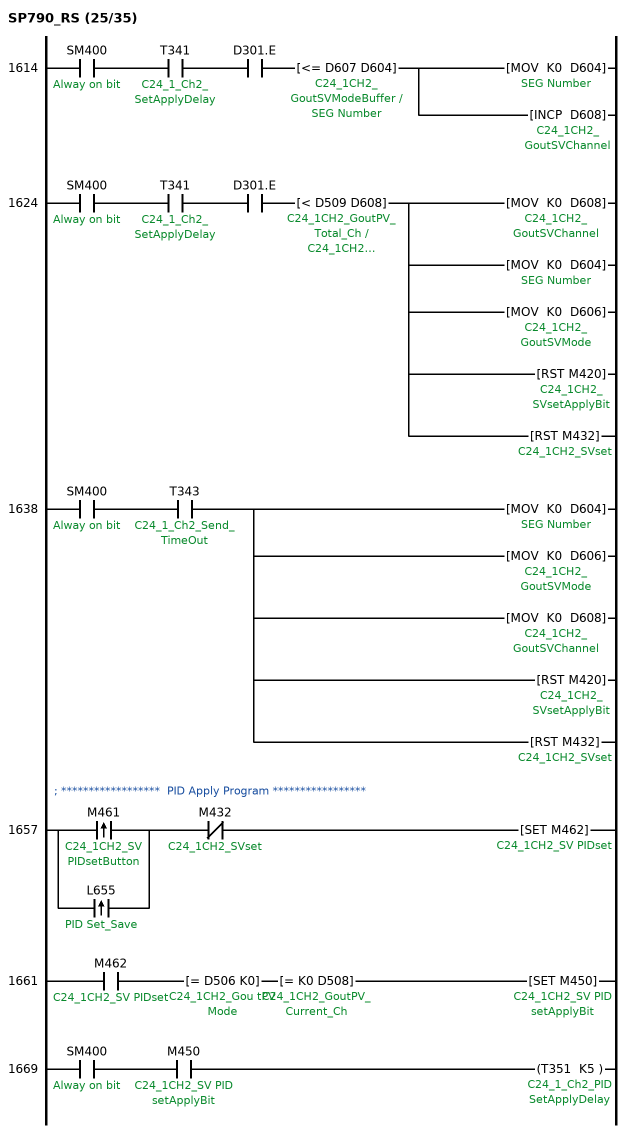
[picture p24: ladder of SP790_RS, rungs at steps 1614 to 1669]
1614  LD      SM400  ; Alway on bit
      AND     T341  ; C24_1_Ch2_SetApplyDelay
      AND     D301.E
      AND<=   D607 D604  ; C24_1CH2_GoutSVModeBuffer / SEG Number
      MOV     K0 D604
      INCP    D608
1624  LD      SM400  ; Alway on bit
      AND     T341  ; C24_1_Ch2_SetApplyDelay
      AND     D301.E
      AND<    D509 D608  ; C24_1CH2_GoutPV_Total_Ch / C24_1CH2_GoutSVChannel
      MOV     K0 D608
      MOV     K0 D604
      MOV     K0 D606
      RST     M420  ; C24_1CH2_SVsetApplyBit
      RST     M432  ; C24_1CH2_SVset
1638  LD      SM400  ; Alway on bit
      AND     T343  ; C24_1_Ch2_Send_TimeOut
      MOV     K0 D604
      MOV     K0 D606
      MOV     K0 D608
      RST     M420  ; C24_1CH2_SVsetApplyBit
      RST     M432  ; C24_1CH2_SVset
; 
; 
; 
; 
; ******************  PID Apply Program *****************
1657  LDP     M461  ; C24_1CH2_SV PIDsetButton
      ORP     L655  ; PID Set_Save
      ANI     M432  ; C24_1CH2_SVset
      SET     M462  ; C24_1CH2_SV PIDset
1661  LD      M462  ; C24_1CH2_SV PIDset
      AND=    D506 K0  ; C24_1CH2_Gou tPV Mode
      AND=    K0 D508  ; C24_1CH2_GoutPV_Current_Ch
      SET     M450  ; C24_1CH2_SV PID setApplyBit
1669  LD      SM400  ; Alway on bit
      AND     M450  ; C24_1CH2_SV PID setApplyBit
      OUT     T351 K5  ; C24_1_Ch2_PID SetApplyDelay
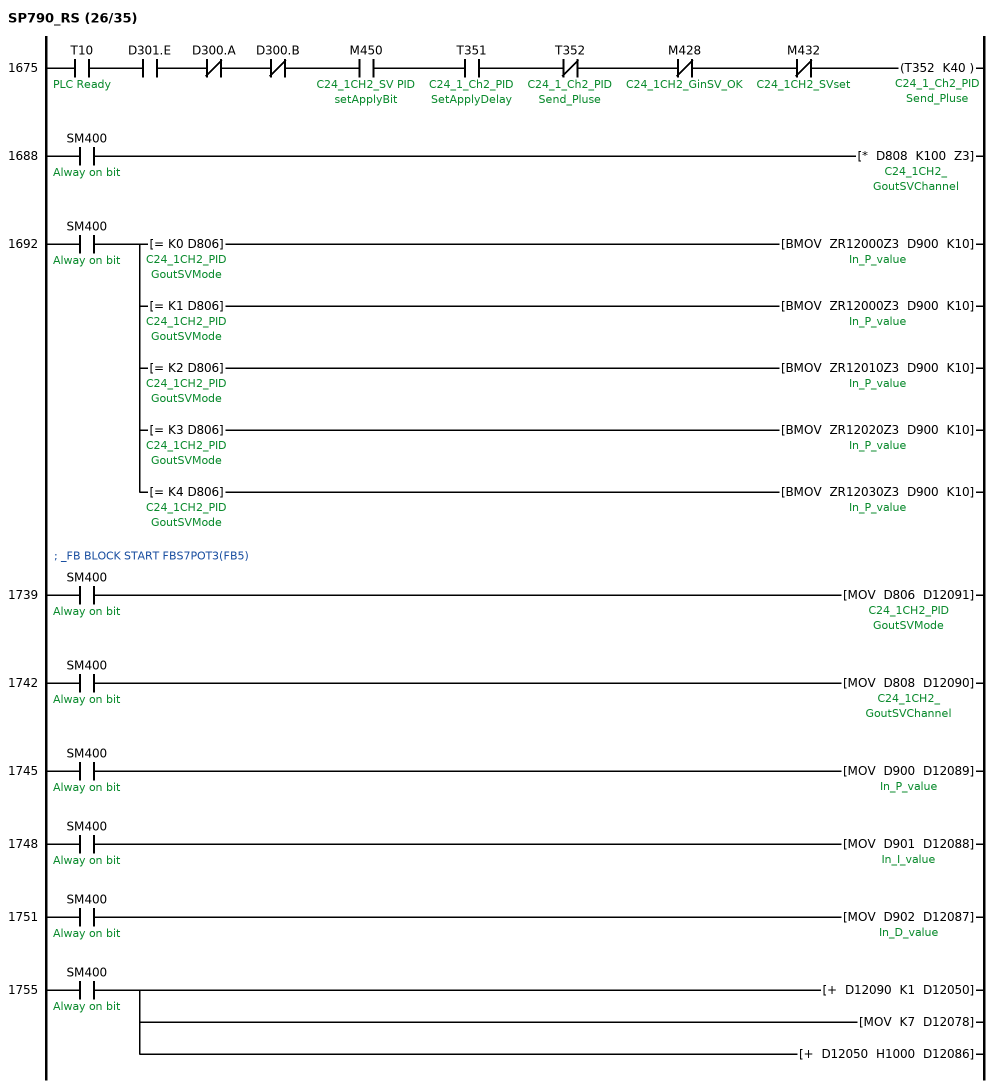
1675  LD      T10  ; PLC Ready
      AND     D301.E
      ANI     D300.A
      ANI     D300.B
      AND     M450  ; C24_1CH2_SV PID setApplyBit
      AND     T351  ; C24_1_Ch2_PID SetApplyDelay
      ANI     T352  ; C24_1_Ch2_PID Send_Pluse
      ANI     M428  ; C24_1CH2_GinSV_OK
      ANI     M432  ; C24_1CH2_SVset
      OUTH    T352 K40  ; C24_1_Ch2_PID Send_Pluse
1688  LD      SM400  ; Alway on bit
      *       D808 K100 Z3  ; C24_1CH2_GoutSVChannel
1692  LD      SM400  ; Alway on bit
      MPS
      AND=    K0 D806  ; C24_1CH2_PID GoutSVMode
      BMOV    ZR12000Z3 D900 K10  ; In_P_value
      MRD
      AND=    K1 D806  ; C24_1CH2_PID GoutSVMode
      BMOV    ZR12000Z3 D900 K10
      MRD
      AND=    K2 D806  ; C24_1CH2_PID GoutSVMode
      BMOV    ZR12010Z3 D900 K10
      MRD
      AND=    K3 D806  ; C24_1CH2_PID GoutSVMode
      BMOV    ZR12020Z3 D900 K10
      MPP
      AND=    K4 D806  ; C24_1CH2_PID GoutSVMode
      BMOV    ZR12030Z3 D900 K10
; _FB BLOCK START FBS7POT3(FB5)
1739  LD      SM400  ; Alway on bit
      MOV     D806 D12091
1742  LD      SM400  ; Alway on bit
      MOV     D808 D12090
1745  LD      SM400  ; Alway on bit
      MOV     D900 D12089
1748  LD      SM400  ; Alway on bit
      MOV     D901 D12088  ; In_I_value
1751  LD      SM400  ; Alway on bit
      MOV     D902 D12087  ; In_D_value
; FB START
1755  LD      SM400  ; Alway on bit
      +       D12090 K1 D12050
      MOV     K7 D12078
      +       D12050 H1000 D12086
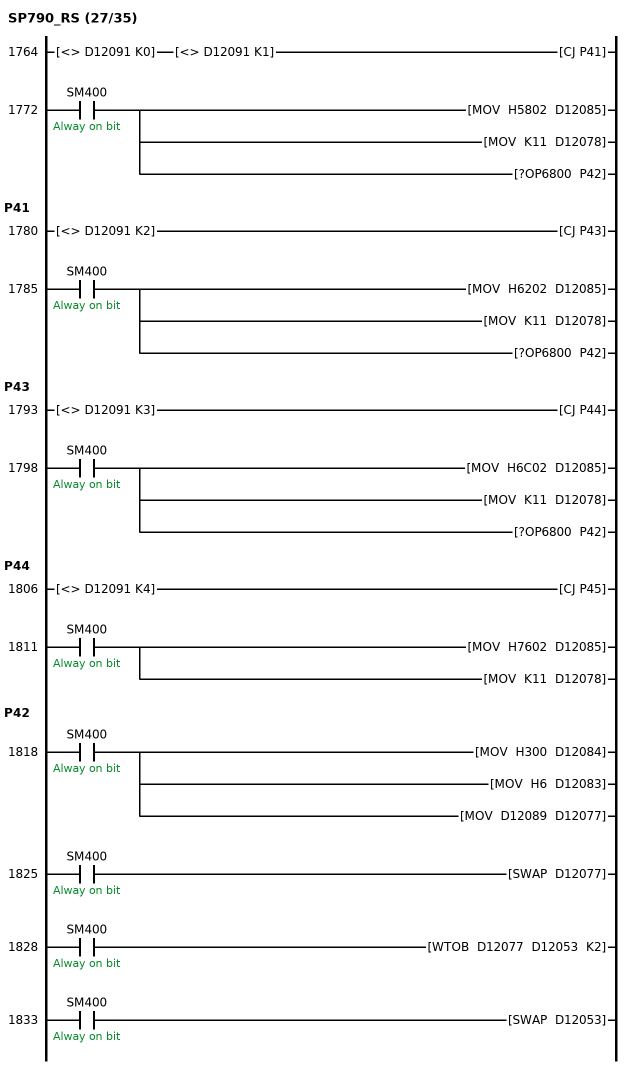
1764  LD<>    D12091 K0
      AND<>   D12091 K1
      CJ      P41
1772  LD      SM400  ; Alway on bit
      MOV     H5802 D12085
      MOV     K11 D12078
      ?OP6800 P42
      P41
1780  LD<>    D12091 K2
      CJ      P43
1785  LD      SM400  ; Alway on bit
      MOV     H6202 D12085
      MOV     K11 D12078
      ?OP6800 P42
      P43
1793  LD<>    D12091 K3
      CJ      P44
1798  LD      SM400  ; Alway on bit
      MOV     H6C02 D12085
      MOV     K11 D12078
      ?OP6800 P42
      P44
1806  LD<>    D12091 K4
      CJ      P45
1811  LD      SM400  ; Alway on bit
      MOV     H7602 D12085
      MOV     K11 D12078
      P45
      P42
1818  LD      SM400  ; Alway on bit
      MOV     H300 D12084
      MOV     H6 D12083
      MOV     D12089 D12077
1825  LD      SM400  ; Alway on bit
      SWAP    D12077
1828  LD      SM400  ; Alway on bit
      WTOB    D12077 D12053 K2
1833  LD      SM400  ; Alway on bit
      SWAP    D12053
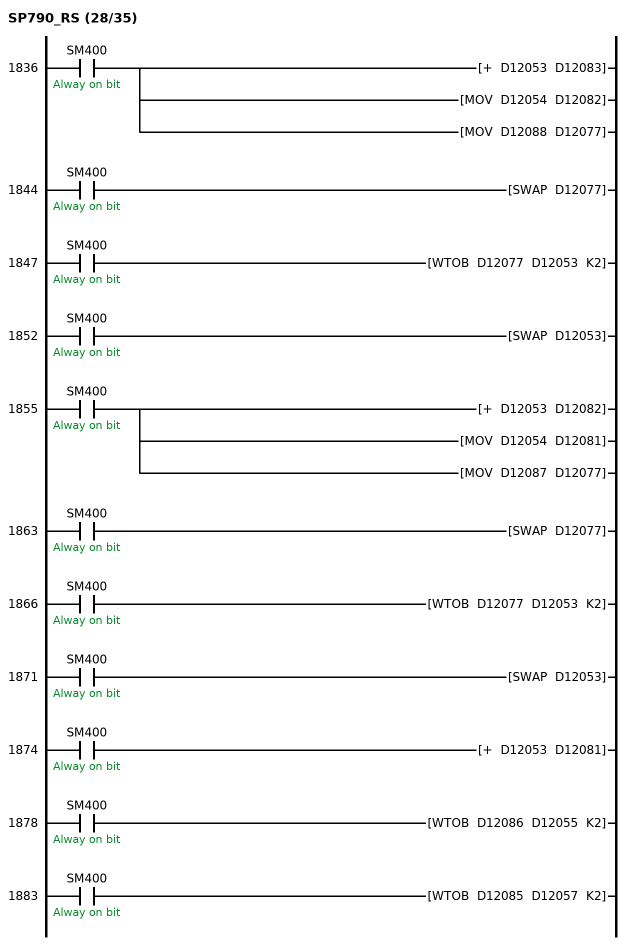
1836  LD      SM400  ; Alway on bit
      +       D12053 D12083
      MOV     D12054 D12082
      MOV     D12088 D12077
1844  LD      SM400  ; Alway on bit
      SWAP    D12077
1847  LD      SM400  ; Alway on bit
      WTOB    D12077 D12053 K2
1852  LD      SM400  ; Alway on bit
      SWAP    D12053
1855  LD      SM400  ; Alway on bit
      +       D12053 D12082
      MOV     D12054 D12081
      MOV     D12087 D12077
1863  LD      SM400  ; Alway on bit
      SWAP    D12077
1866  LD      SM400  ; Alway on bit
      WTOB    D12077 D12053 K2
1871  LD      SM400  ; Alway on bit
      SWAP    D12053
1874  LD      SM400  ; Alway on bit
      +       D12053 D12081
1878  LD      SM400  ; Alway on bit
      WTOB    D12086 D12055 K2
1883  LD      SM400  ; Alway on bit
      WTOB    D12085 D12057 K2
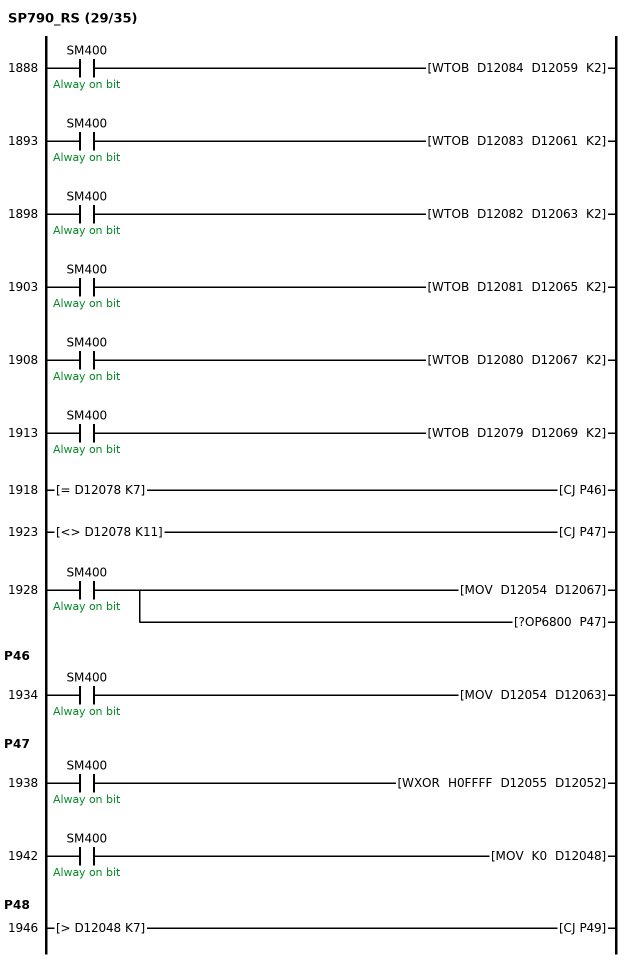
1888  LD      SM400  ; Alway on bit
      WTOB    D12084 D12059 K2
1893  LD      SM400  ; Alway on bit
      WTOB    D12083 D12061 K2
1898  LD      SM400  ; Alway on bit
      WTOB    D12082 D12063 K2
1903  LD      SM400  ; Alway on bit
      WTOB    D12081 D12065 K2
1908  LD      SM400  ; Alway on bit
      WTOB    D12080 D12067 K2
1913  LD      SM400  ; Alway on bit
      WTOB    D12079 D12069 K2
1918  LD=     D12078 K7
      CJ      P46
1923  LD<>    D12078 K11
      CJ      P47
1928  LD      SM400  ; Alway on bit
      MOV     D12054 D12067
      ?OP6800 P47
      P46
1934  LD      SM400  ; Alway on bit
      MOV     D12054 D12063
      P47
1938  LD      SM400  ; Alway on bit
      WXOR    H0FFFF D12055 D12052
1942  LD      SM400  ; Alway on bit
      MOV     K0 D12048
      P48
1946  LD>     D12048 K7
      CJ      P49
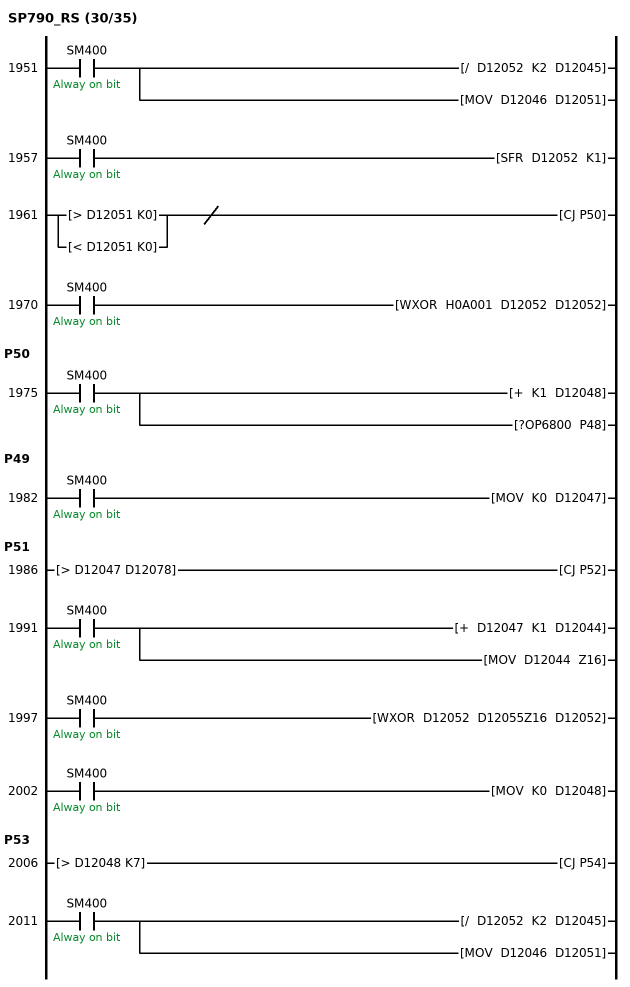
1951  LD      SM400  ; Alway on bit
      /       D12052 K2 D12045
      MOV     D12046 D12051
1957  LD      SM400  ; Alway on bit
      SFR     D12052 K1
1961  LD>     D12051 K0
      OR<     D12051 K0
      INV
      CJ      P50
1970  LD      SM400  ; Alway on bit
      WXOR    H0A001 D12052 D12052
      P50
1975  LD      SM400  ; Alway on bit
      +       K1 D12048
      ?OP6800 P48
      P49
1982  LD      SM400  ; Alway on bit
      MOV     K0 D12047
      P51
1986  LD>     D12047 D12078
      CJ      P52
1991  LD      SM400  ; Alway on bit
      +       D12047 K1 D12044
      MOV     D12044 Z16
1997  LD      SM400  ; Alway on bit
      WXOR    D12052 D12055Z16 D12052
2002  LD      SM400  ; Alway on bit
      MOV     K0 D12048
      P53
2006  LD>     D12048 K7
      CJ      P54
2011  LD      SM400  ; Alway on bit
      /       D12052 K2 D12045
      MOV     D12046 D12051
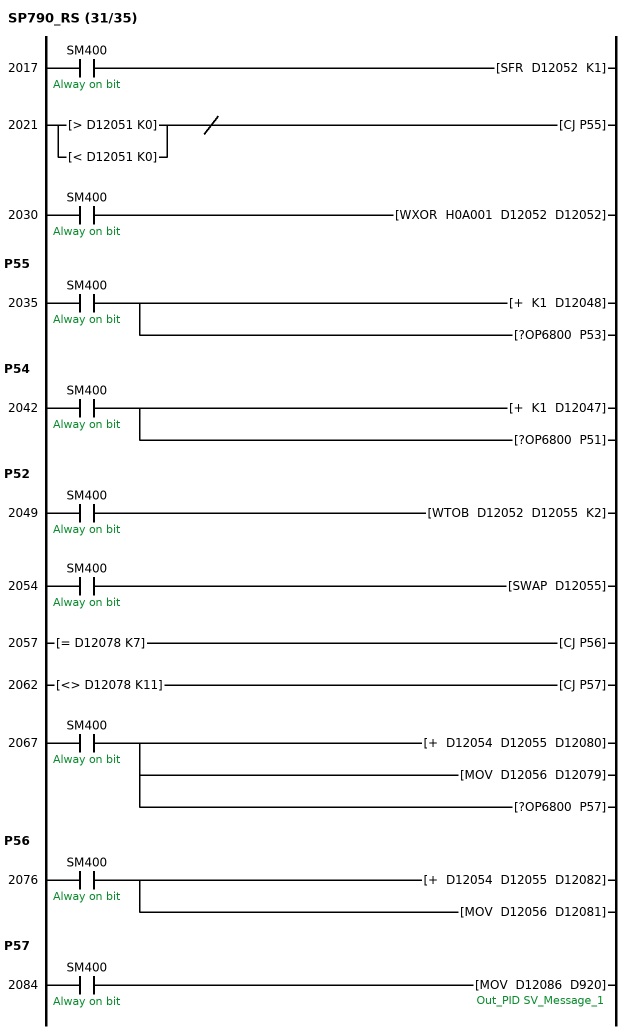
2017  LD      SM400  ; Alway on bit
      SFR     D12052 K1
2021  LD>     D12051 K0
      OR<     D12051 K0
      INV
      CJ      P55
2030  LD      SM400  ; Alway on bit
      WXOR    H0A001 D12052 D12052
      P55
2035  LD      SM400  ; Alway on bit
      +       K1 D12048
      ?OP6800 P53
      P54
2042  LD      SM400  ; Alway on bit
      +       K1 D12047
      ?OP6800 P51
      P52
2049  LD      SM400  ; Alway on bit
      WTOB    D12052 D12055 K2
2054  LD      SM400  ; Alway on bit
      SWAP    D12055
2057  LD=     D12078 K7
      CJ      P56
2062  LD<>    D12078 K11
      CJ      P57
2067  LD      SM400  ; Alway on bit
      +       D12054 D12055 D12080
      MOV     D12056 D12079
      ?OP6800 P57
      P56
2076  LD      SM400  ; Alway on bit
      +       D12054 D12055 D12082
      MOV     D12056 D12081
      P57
; FB END
2084  LD      SM400  ; Alway on bit
      MOV     D12086 D920  ; Out_PID SV_Message_1
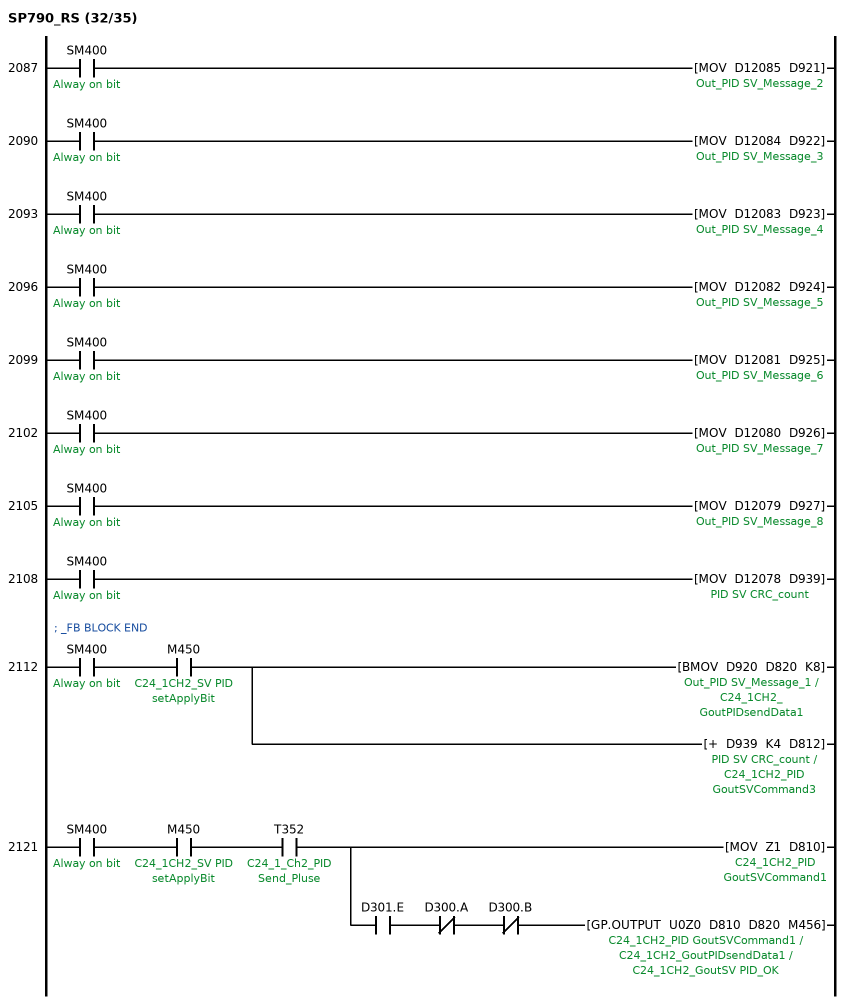
2087  LD      SM400  ; Alway on bit
      MOV     D12085 D921  ; Out_PID SV_Message_2
2090  LD      SM400  ; Alway on bit
      MOV     D12084 D922  ; Out_PID SV_Message_3
2093  LD      SM400  ; Alway on bit
      MOV     D12083 D923  ; Out_PID SV_Message_4
2096  LD      SM400  ; Alway on bit
      MOV     D12082 D924  ; Out_PID SV_Message_5
2099  LD      SM400  ; Alway on bit
      MOV     D12081 D925  ; Out_PID SV_Message_6
2102  LD      SM400  ; Alway on bit
      MOV     D12080 D926  ; Out_PID SV_Message_7
2105  LD      SM400  ; Alway on bit
      MOV     D12079 D927  ; Out_PID SV_Message_8
2108  LD      SM400  ; Alway on bit
      MOV     D12078 D939
; _FB BLOCK END
2112  LD      SM400  ; Alway on bit
      AND     M450  ; C24_1CH2_SV PID setApplyBit
      BMOV    D920 D820 K8  ; C24_1CH2_GoutPIDsendData1
      +       D939 K4 D812  ; C24_1CH2_PID GoutSVCommand3
2121  LD      SM400  ; Alway on bit
      AND     M450  ; C24_1CH2_SV PID setApplyBit
      AND     T352  ; C24_1_Ch2_PID Send_Pluse
      MOV     Z1 D810  ; C24_1CH2_PID GoutSVCommand1
      AND     D301.E
      ANI     D300.A
      ANI     D300.B
      GP.OUTPUT U0Z0 D810 D820 M456  ; C24_1CH2_GoutSV PID_OK
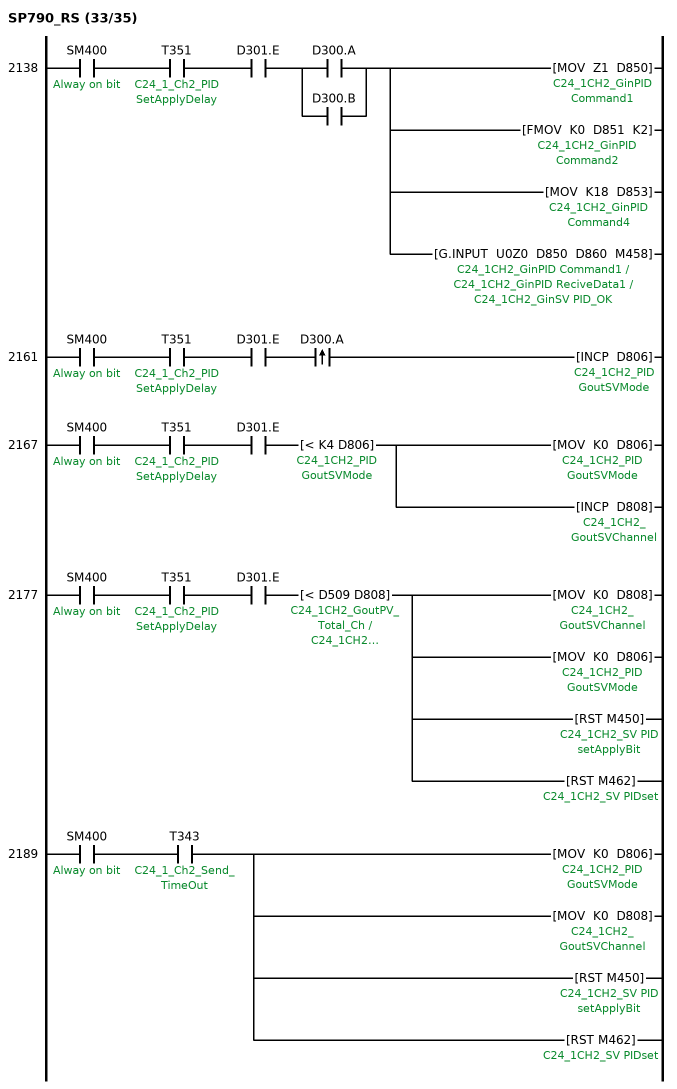
2138  LD      SM400  ; Alway on bit
      AND     T351  ; C24_1_Ch2_PID SetApplyDelay
      AND     D301.E
      LD      D300.A
      OR      D300.B
      ANB
      MOV     Z1 D850  ; C24_1CH2_GinPID Command1
      FMOV    K0 D851 K2  ; C24_1CH2_GinPID Command2
      MOV     K18 D853  ; C24_1CH2_GinPID Command4
      G.INPUT U0Z0 D850 D860 M458  ; C24_1CH2_GinPID ReciveData1 / C24_1CH2_GinSV PID_OK
2161  LD      SM400  ; Alway on bit
      AND     T351  ; C24_1_Ch2_PID SetApplyDelay
      AND     D301.E
      ANDP    D300.A
      INCP    D806
2167  LD      SM400  ; Alway on bit
      AND     T351  ; C24_1_Ch2_PID SetApplyDelay
      AND     D301.E
      AND<    K4 D806  ; C24_1CH2_PID GoutSVMode
      MOV     K0 D806
      INCP    D808
2177  LD      SM400  ; Alway on bit
      AND     T351  ; C24_1_Ch2_PID SetApplyDelay
      AND     D301.E
      AND<    D509 D808  ; C24_1CH2_GoutPV_Total_Ch / C24_1CH2_GoutSVChannel
      MOV     K0 D808
      MOV     K0 D806
      RST     M450  ; C24_1CH2_SV PID setApplyBit
      RST     M462  ; C24_1CH2_SV PIDset
2189  LD      SM400  ; Alway on bit
      AND     T343  ; C24_1_Ch2_Send_TimeOut
      MOV     K0 D806
      MOV     K0 D808
      RST     M450  ; C24_1CH2_SV PID setApplyBit
      RST     M462  ; C24_1CH2_SV PIDset
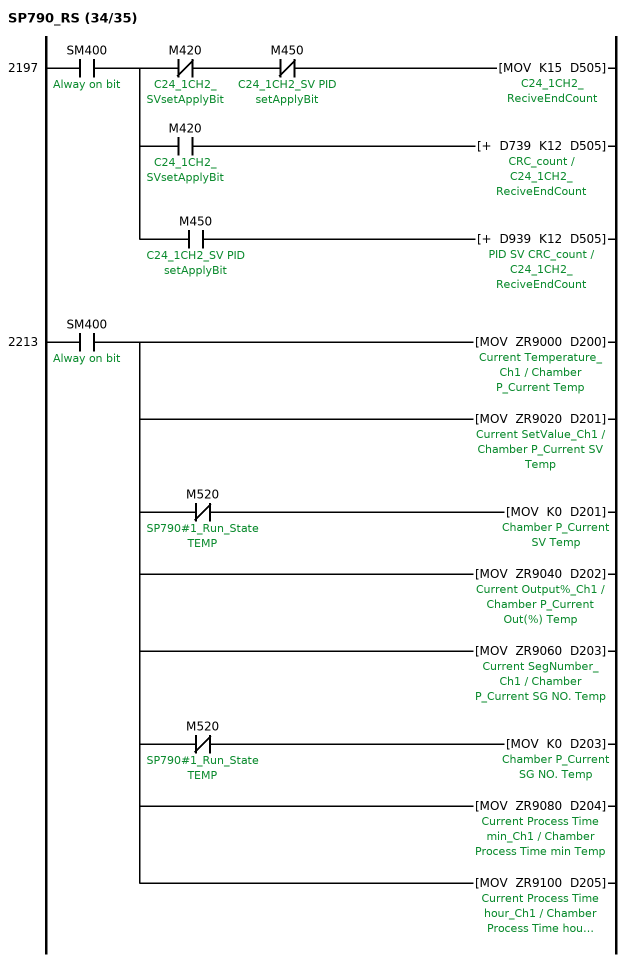
2197  LD      SM400  ; Alway on bit
      MPS
      ANI     M420  ; C24_1CH2_SVsetApplyBit
      ANI     M450  ; C24_1CH2_SV PID setApplyBit
      MOV     K15 D505
      MRD
      AND     M420  ; C24_1CH2_SVsetApplyBit
      +       D739 K12 D505
      MPP
      AND     M450  ; C24_1CH2_SV PID setApplyBit
      +       D939 K12 D505
2213  LD      SM400  ; Alway on bit
      MOV     ZR9000 D200  ; Current Temperature_Ch1 / Chamber P_Current Temp
      MOV     ZR9020 D201  ; Current SetValue_Ch1 / Chamber P_Current SV Temp
      MPS
      ANI     M520  ; SP790#1_Run_State TEMP
      MOV     K0 D201
      MPP
      MOV     ZR9040 D202  ; Current Output%_Ch1 / Chamber P_Current Out(%) Temp
      MOV     ZR9060 D203  ; Current SegNumber_Ch1 / Chamber P_Current SG NO. Temp
      MPS
      ANI     M520  ; SP790#1_Run_State TEMP
      MOV     K0 D203
      MPP
      MOV     ZR9080 D204  ; Current Process Time min_Ch1 / Chamber Process Time min Temp
      MOV     ZR9100 D205  ; Current Process Time hour_Ch1 / Chamber Process Time hour Temp
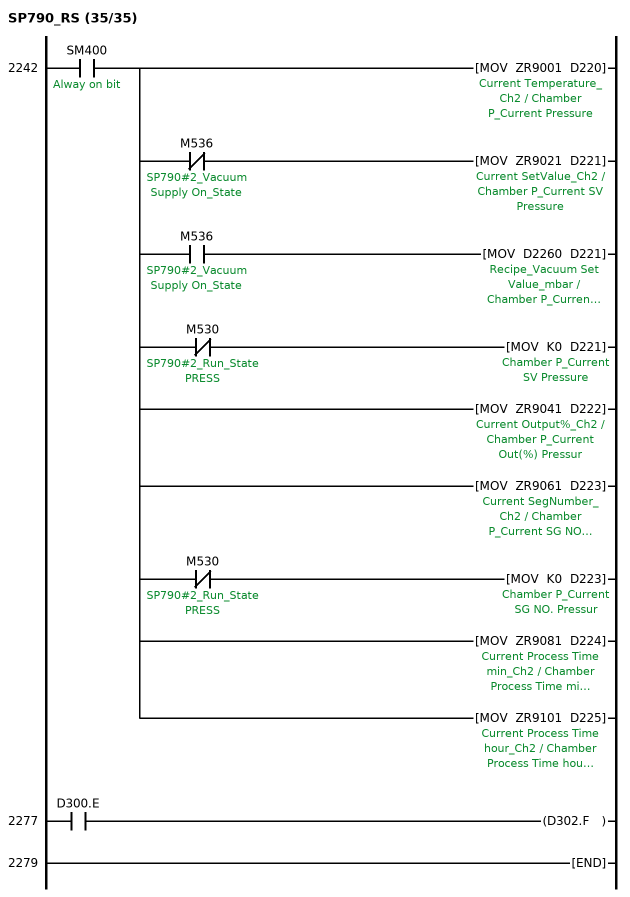
2242  LD      SM400  ; Alway on bit
      MOV     ZR9001 D220  ; Current Temperature_Ch2 / Chamber P_Current Pressure
      MPS
      ANI     M536  ; SP790#2_Vacuum Supply On_State
      MOV     ZR9021 D221  ; Current SetValue_Ch2 / Chamber P_Current SV Pressure
      MRD
      AND     M536  ; SP790#2_Vacuum Supply On_State
      MOV     D2260 D221  ; Recipe_Vacuum Set Value_mbar
      MRD
      ANI     M530  ; SP790#2_Run_State PRESS
      MOV     K0 D221
      MPP
      MOV     ZR9041 D222  ; Current Output%_Ch2 / Chamber P_Current Out(%) Pressur
      MOV     ZR9061 D223  ; Current SegNumber_Ch2 / Chamber P_Current SG NO. Pressur
      MPS
      ANI     M530  ; SP790#2_Run_State PRESS
      MOV     K0 D223
      MPP
      MOV     ZR9081 D224  ; Current Process Time min_Ch2 / Chamber Process Time min Pressur
      MOV     ZR9101 D225  ; Current Process Time hour_Ch2 / Chamber Process Time hour Pressu
2277  LD      D300.E
      OUT     D302.F
2279  END
END_PROGRAM
